(* CODESYS project sensores_v2_2_14.library
   Company: Teknike
   Version: 2.2.14
   DefaultNamespace: Teknike_Sensores
   Title: Sensores
   Placeholder: Teknike_Sensores
   Author: Tiago B. Cunico
   DocFormat: reStructuredText

Project tree, tasks and I/O mapping:
  libraries: BASIC, 3.31 (OSCAT); Tc2_ModbusRTU, * (Beckhoff Automation GmbH); Tc2_Standard, * (Beckhoff Automation GmbH); Tc2_System, * (Beckhoff Automation GmbH); Tc2_TcpIp, * (Beckhoff Automation GmbH); Tc2_Utilities, * (Beckhoff Automation GmbH); Tc3_Database, * (Beckhoff Automation GmbH); Tc3_Module, * (Beckhoff Automation GmbH); Geral, * (Teknike); TwinCAT Dynamic String Kit, * (FisoThemes)
  DUTs/
  Fbs/
    Analogica/
      Duts/
        data type Config_ST_SensorAnalogicos
        data type en_ST_SensorAnalogico
        data type sa_ST_SensorAnalogico
        data type st_SensorAnalogico
      function block FB_SensorAnalogico [ST]: AjeitaEntrada, AjeitaSaida
    Digital/
      SensorDigital/
        Duts/
          data type Config_ST_SensorDigital
          data type en_ST_SensorDigital
          data type ENUM_StatusSensor
          data type sa_ST_SensorDigital
          data type st_LeConfigSensorNoBanco
          data type st_SensorDigital
        function block FB_SensorDigital [ST]: FB_init, TamanhoCaixa
    Rede/
      322_485_Novus/
        Duts/
          data type entrada_N322_485_Novus
          data type Saida_N322_485_Novus
          data type st_N322_485_Novus
        function block N322_485_Novus [ST]
      RFID/
        function block FB_LeitorRFID_ViaOnda [ST]
        data type st_LeitorRFID_ViaOnda
      RTH_485_Novus/
        Duts/
          data type Config_RTH_485_Novus
          data type dt_RTH_485_Novus
          data type entrada_RTH_485_Novus
          data type Saida_RTH_485_Novus
        function block RTH_485_Novus [ST]
      SR2000/
        duts/
          data type ST_SR2000
          data type ST_SR2000_Config
          data type ST_SR2000_Entradas_Bloco
          data type ST_SR2000_Entradas_Dispositivo
          data type ST_SR2000_Saidas_Bloco
          data type ST_SR2000_Saidas_Dispositivo
        function F_AjeitaStringLeitor [ST]
        function block FB_SR2000 [ST]: AjustaEntrada, AjustaSaida, ContagemFalha, RequisitaDados, Status, TempoLeitura, TrabalhaResultado, Trigger
  GVLs/
    global variables GVL_Teste
  POUs/
    global variables GVL_BlibliotecaSensores
    program MAIN [ST]: ACT, Digital, SensorAnalogico
    program ValidaLicensa [ST]: Licensas
  Project Information/
    function F_GetCompany [ST]
    function F_GetTitle [ST]
    function F_GetVersion [ST]
  Version/
    global variables Global_Version
  VISUs/
*)

// Fbs/Analogica/Duts/Config_ST_SensorAnalogicos
TYPE Config_ST_SensorAnalogicos :
STRUCT PERSISTENT RETAIN
	rMinEntrada : REAL := 0; // valor minimo da entrada, normalmente 0
	rMaxEntrada : REAL := 32767; // valor maximo da entrada, normalmente 32767
	rMinSaida 	: REAL := 0; //minimo saida, normalmente 0
	rMaxSaida 	: REAL; // valor final, esse depende muito com o sensor
	iTempoFiltro: UDINT; // em ms
	sNome_Funcao: STRING;
	rOffset		: REAL; // offset direto na saida
		
	xForcaValor		: BOOL;				// ai ignora o valor que ta calculando e usa o valor que o cara setar
	rValorForcado	: REAL;				// valor que vai ser forçado
END_STRUCT
END_TYPE

// Fbs/Analogica/Duts/en_ST_SensorAnalogico
TYPE en_ST_SensorAnalogico :
	STRUCT
		iEntrada	: INT;	// valor vindo do sensor	
		i			: INT;	// Index para a IHM
	END_STRUCT
END_TYPE

// Fbs/Analogica/Duts/sa_ST_SensorAnalogico
TYPE sa_ST_SensorAnalogico :
	STRUCT
		rValor : REAL; // valor filtrado
		xPossivelFalha : BOOL; // se ficar mais de x tempo no no fim de escala ou no inicio dela é pq provavelmente deu pau
	END_STRUCT
END_TYPE

// Fbs/Analogica/Duts/st_SensorAnalogico
TYPE st_SensorAnalogico :
	STRUCT
		en		: en_ST_SensorAnalogico;
		config	: Config_ST_SensorAnalogicos;
		sa		: sa_ST_SensorAnalogico;
	END_STRUCT
END_TYPE

// Fbs/Digital/SensorDigital/Duts/Config_ST_SensorDigital
TYPE Config_ST_SensorDigital :
STRUCT RETAIN PERSISTENT
	xNF:		BOOL;
	rTmpOn:		REAL;
	rTmpOff:	REAL;
	sNome_Funcao: STRING;
END_STRUCT
END_TYPE

// Fbs/Digital/SensorDigital/Duts/en_ST_SensorDigital
TYPE en_ST_SensorDigital :
	STRUCT
		xSinalSensor	: BOOL;
		xResetContagem	: BOOL;
		i				: INT; // Index para a IHM	
		rVeloEsteira	: REAL;
	END_STRUCT
END_TYPE

// Fbs/Digital/SensorDigital/Duts/ENUM_StatusSensor
//{attribute 'qualified_only'}
//{attribute 'strict'}
TYPE ENUM_StatusSensor :
	(
		OBJETO_AUSENTE		:= 0,
		DETECTANDO_OBJETO	:= 1,
		OBJETO_PRESENTE		:= 2,
		DETECTANDO_AUSENCIA	:= 3
	);
END_TYPE

// Fbs/Digital/SensorDigital/Duts/sa_ST_SensorDigital
TYPE sa_ST_SensorDigital :
	STRUCT
		xObjPresente	: BOOL;
		uiContagem		: UINT;
		eStatus			: ENUM_StatusSensor;
		rTamanhoCaixa	: REAL; // tamanho da caixa em milimetros
	END_STRUCT
END_TYPE

// Fbs/Digital/SensorDigital/Duts/st_LeConfigSensorNoBanco
TYPE st_LeConfigSensorNoBanco :
	STRUCT
		Sensor		: T_ULARGE_INTEGER;
		Tag			: STRING(80);
		Funcao		: STRING(80);
		Timestamp	: DT;
	END_STRUCT
END_TYPE

// Fbs/Digital/SensorDigital/Duts/st_SensorDigital
TYPE st_SensorDigital :
	STRUCT
		en		: en_ST_SensorDigital;
		config	: Config_ST_SensorDigital;
		sa		: sa_ST_SensorDigital;
		Banco	: st_LeConfigSensorNoBanco;
	END_STRUCT
END_TYPE

// Fbs/Rede/322_485_Novus/Duts/entrada_N322_485_Novus
TYPE entrada_N322_485_Novus :
	STRUCT
		xComeca		: BOOL;
		iEndereco	: INT;	//endereço dele na rede
		i			: INT;	// Index para a IHM
		sNomeFuncao	: STRING;
		xForcaFalor : BOOL;
		rValorForcado : REAL;
		rOffset : REAL;
	END_STRUCT
END_TYPE

// Fbs/Rede/322_485_Novus/Duts/Saida_N322_485_Novus
TYPE Saida_N322_485_Novus :
	STRUCT
		xOcupado			: BOOL;
		xTerminei			: BOOL;
		rTemp				: REAL;
		xOnline				: BOOL;
		UltimoModbusErro	: MODBUS_ERRORS;
	END_STRUCT
END_TYPE

// Fbs/Rede/322_485_Novus/Duts/st_N322_485_Novus
TYPE st_N322_485_Novus :
	STRUCT
		en	: entrada_N322_485_Novus;
		sa	: Saida_N322_485_Novus;
	END_STRUCT
END_TYPE

// Fbs/Rede/RFID/st_LeitorRFID_ViaOnda
TYPE st_LeitorRFID_ViaOnda :
STRUCT
	xConecta : BOOL;	
	ip : T_IPv4Addr;
	xNovoResultado : BOOL;
	sTag : STRING;
	iTag : INT;
	xOnline : BOOL; //
END_STRUCT
END_TYPE

// Fbs/Rede/RTH_485_Novus/Duts/Config_RTH_485_Novus
TYPE Config_RTH_485_Novus :
STRUCT PERSISTENT RETAIN
	iEndereco 			: INT;
	iModoIndicacao		: INT;
	xUnidadeDeMedida	: BOOL;
	xBloqueiaConfigBT	: BOOL;
	rOffSetTemperatura	: REAL;
	rOffSetUmidade		: REAL;
	uiValorErro			: UINT;
END_STRUCT
END_TYPE

// Fbs/Rede/RTH_485_Novus/Duts/dt_RTH_485_Novus
TYPE dt_RTH_485_Novus :
	STRUCT
		en		: entrada_RTH_485_Novus;
		Config	: Config_RTH_485_Novus;
		sa		: Saida_RTH_485_Novus;
	END_STRUCT
END_TYPE

// Fbs/Rede/RTH_485_Novus/Duts/entrada_RTH_485_Novus
TYPE entrada_RTH_485_Novus :
	STRUCT
		xComeca			: BOOL;
		xEscreve		: BOOL;
		xAtualizaTudo	: BOOL;
		i				: INT; // Index para a IHM
	END_STRUCT
END_TYPE

// Fbs/Rede/RTH_485_Novus/Duts/Saida_RTH_485_Novus
TYPE Saida_RTH_485_Novus :
	STRUCT
		xTerminei : BOOL;

		rTemp					: REAL;
		rUmidade				: REAL;
		rPontoDeOrvalho			: REAL;
		iModoIndicacaoAtual		: INT;
		xUnidadeDeMedidaAtual	: BOOL;
		xHabilitaConfigBTAtual	: BOOL;
		rOffSetTemperaturaAtual	: REAL;
		rOffSetUmidadeAtual		: REAL;
		uiValorErroAtual		: UINT;
		xOnline					: BOOL;
		UltimoModbusErro		: ST_ModbusErrorDiagnostics;
	END_STRUCT
END_TYPE

// Fbs/Rede/SR2000/duts/ST_SR2000
TYPE ST_SR2000 :
	STRUCT
		En	: ST_SR2000_Entradas_Bloco;
		Sa	: ST_SR2000_Saidas_Bloco;
		Config : ST_SR2000_Config;
		

		En_D	AT %I*	: ST_SR2000_Entradas_Dispositivo;
		Sa_D	AT %Q*	: ST_SR2000_Saidas_Dispositivo;
	END_STRUCT
END_TYPE

// Fbs/Rede/SR2000/duts/ST_SR2000_Config
TYPE ST_SR2000_Config :
	STRUCT RETAIN PERSISTENT
		iIgnoraInicio : INT;
		iQuantosCharLe : INT;
	END_STRUCT
END_TYPE

// Fbs/Rede/SR2000/duts/ST_SR2000_Entradas_Bloco
TYPE ST_SR2000_Entradas_Bloco :
	STRUCT
		xLiga					: BOOL;
		xHabilitaAutoTrigger	: BOOL := true;
		xBtTriggerManual		: BOOL;
		xTrigManualCiclico		: BOOL;
		xSinalTrigAutomatico	: BOOL;
		xReset					: BOOL;
		sNome_Funcao			: STRING;
	END_STRUCT
END_TYPE

// Fbs/Rede/SR2000/duts/ST_SR2000_Entradas_Dispositivo
TYPE ST_SR2000_Entradas_Dispositivo :
	STRUCT

		State : UINT;

		xError					: BIT;
		xResultDataAvailable	: BIT;
		xResultDataStrobe		: BIT;

		xBufferOverflowError	: BIT;
		xGeneralError			: BIT;
		xBusy					: BIT;
		xTriggerBusy			: BIT;
		xLockBusy				: BIT;
		xModeBusy				: BIT;
		xErrBusy				: BIT;

		xREADY : BIT;

		xReadComplete				: BIT;
		xPresetComplete				: BIT;
		xRegisterPresetDataComplete	: BIT;
		xTuneComplete				: BIT;
		xBloadComplete				: BIT;

		xEXTRequestComplete			: BIT;
		xReadingFailure				: BIT;
		xPresetFailure				: BIT;
		xRegisterPresetDataFailure	: BIT;
		xTuneFailure				: BIT;
		xBloadFailure				: BIT;

		xEXTRequestFailure	: BIT;
		xIN1Status			: BIT;
		xIN2Status			: BIT;

		xOUT1Status	: BIT;
		xOUT2Status	: BIT;
		xOUT3Status	: BIT;

		xUnstable				: BIT;
		xMatchingLevelUnstable	: BIT;
		xISO_IEC15415Unstable	: BIT;
		xAIM_DPMUnstable		: BIT;
		xSAE_AS9132Unstable		: BIT;
		xISO_IEC15416Unstable	: BIT;

		uiMatchingLevel					: UINT;
		uiISO_IEC15415Grade				: UINT;
		uiAIM_DPMGrade					: UINT;
		uiISO_IEC15416Grade				: UINT;
		uiReadResultCode				: UINT;
		uiPresetResultCode				: UINT;
		uiRegisterPresetDataResultCode	: UINT;
		uiTuneResultCode				: UINT;
		uiBloadResultCode				: UINT;

		EXTRequestResultCode	: UINT;
		uiGeneralErrorCode		: UINT;
		uiSlaveID				: UINT;
		uiResultDataReadyCount	: UINT;
		uiResultDataUpdateCount	: UINT;
		uiMasterTriggerCount	: UINT;
		uiReadDataSize			: UINT;
		arResultData			: ARRAY[0..128] OF BYTE;

	END_STRUCT
END_TYPE

// Fbs/Rede/SR2000/duts/ST_SR2000_Saidas_Bloco
TYPE ST_SR2000_Saidas_Bloco :
	STRUCT

		xLeitorEmFalha	: BOOL;
		xLeitorPronto	: BOOL;
		xFalhaRede		: BOOL;
		ReadRequest		: BOOL;
		xNovoResultado	: BOOL;
		xFalhaLeitura	: BOOL;
		xNovosDados		: BOOL;
		sCodigoBruto	: STRING;
		sCodigo			: STRING;

		matchPorcentagem	: INT;
		NotaIsoIEC15415		: STRING;
		NotaIsoIEC15416		: STRING;
		NotaAimDPM			: STRING;

		uiTrigsTotais		: UINT;
		uiSucessoTotais		: UINT;
		uiFalhasTotais		: UINT;
		AcertoPorcentagem	: REAL;

		xSinalDeLiga : BOOL;
		
		sTempoTotalDeLeitura : STRING;
		sMediaTempoTotalDeLeitura : STRING;
	END_STRUCT
END_TYPE

// Fbs/Rede/SR2000/duts/ST_SR2000_Saidas_Dispositivo
TYPE ST_SR2000_Saidas_Dispositivo :
	STRUCT

		ctrl : UINT;

		ResultDataLatch				: BIT;
		ErrorClear					: BIT;
		ReadRequest					: BIT;
		PresetRequest				: BIT;
		RegisterPresetDataRequest	: BIT;
		TuneRequest					: BIT;
		BloadRequest				: BIT;

		ReadCompleteClear				: BIT;
		PresetCompleteClear				: BIT;
		RegisterPresetDataCompleteClear	: BIT;
		TuneCompleteClear				: BIT;
		BloadCompleteClear				: BIT;

		EXTRequestCompleteClear : BIT;

		BankNumber : UINT;

		UserDataSize	: UINT;
		UserData		: ARRAY[0..63] OF BYTE;
	END_STRUCT
END_TYPE

// GVLs/GVL_Teste
//{attribute 'qualified_only'}
VAR_GLOBAL PERSISTENT RETAIN

	stDigitaisss : st_SensorDigital;

	RTU : st_N322_485_Novus;

END_VAR

// POUs/GVL_BlibliotecaSensores
//{attribute 'qualified_only'}
VAR_GLOBAL
    {attribute 'hide'} 
	{attribute 'tc_no_symbol'}
	xLicensaValida1616848sdfs : BOOL;
	LicensaValida : BOOL;
	STCheckLicense : ST_CheckLicense;
END_VAR

// Version/Global_Version
{attribute 'TcGenerated'}
{attribute 'no-analysis'}
{attribute 'linkalways'}
// This function has been automatically generated from the project information.
VAR_GLOBAL CONSTANT
	{attribute 'const_non_replaced'}
	stLibVersion_Sensores : ST_LibVersion := (iMajor := 2, iMinor := 2, iBuild := 14, iRevision := 0, nFlags := 0, sVersion := '2.2.14');
END_VAR

// Fbs/Analogica/FB_SensorAnalogico
FUNCTION_BLOCK FB_SensorAnalogico
VAR_IN_OUT
	stAna : st_SensorAnalogico;
END_VAR
VAR_INPUT

	iEntrada		: INT;				// valor vindo do sensor	
	rMinEntrada		: REAL	:= 0;		// valor minimo da entrada, normalmente 0
	rMaxEntrada		: REAL	:= 32767;	// valor maximo da entrada, normalmente 32767
	rMinSaida		: REAL	:= 0;		// minimo saida, normalmente 0
	rMaxSaida		: REAL;				// valor final, esse depende muito com o sensor
	iTempoFiltro	: UDINT;			// em ms
	sNome_Funcao	: STRING;
	rOffset			: REAL; 			// offset direto na saida
	
	xForcaValor		: BOOL;				// ai ignora o valor que ta calculando e usa o valor que o cara setar
	rValorForcado	: REAL;				// valor que vai ser forçado

END_VAR
VAR_OUTPUT
	rValor : REAL; // valor filtrado
	xPossivelFalha : BOOL; // se ficar mais de x tempo no no fim de escala ou no inicio dela é pq provavelmente deu pau
END_VAR
VAR
	filtro	: BASIC.FT_PT1 (*Filter_PT1*) ;
	rAux	: REAL;
	
	tonFalha : TON;
	
	stAnaAnterior : st_SensorAnalogico;
END_VAR

IF xLicensaValida1616848sdfs THEN
	
	AjeitaEntrada();
	
	// transforma de inteiro pra real 
	rAux := BASIC.SCALE_R
		(
			X := iEntrada,
				I_LO := rMinEntrada,
				I_HI := rMaxEntrada,
				O_LO := rMinSaida,
				O_HI := rMaxSaida);
	
	// aplica um filtro de primeira ordem	
	
	//sanitizando entrada pra nao dar execção na bliblioteca do oscat
	IF iTempoFiltro < 5 AND iTempoFiltro <> 0 THEN
		filtro(in := rAux, T := UDINT_TO_TIME(0), K := 1, out => rValor);
	ELSE
		filtro(in := rAux, T := UDINT_TO_TIME(iTempoFiltro), K := 1, out => rValor);
	END_IF
	
	tonFalha(IN:= iEntrada = rMinEntrada OR iEntrada = rMaxEntrada, PT:= T#5M, Q=> xPossivelFalha, ET=> );
	
	rValor := rValor + rOffset;

	IF xForcaValor THEN
		rValor := rValorForcado;
	END_IF
	
	AjeitaSaida();
ELSE
	ValidaLicensa();
END_IF

ACTION AjeitaEntrada:





IF stAna.en.iEntrada <> stAnaAnterior.en.iEntrada THEN
	iEntrada := stAna.en.iEntrada;
END_IF
IF stAna.en.iEntrada <> iEntrada THEN
	stAna.en.iEntrada := iEntrada;
END_IF


IF stAna.config.rMinEntrada <> stAnaAnterior.config.rMinEntrada THEN
	rMinEntrada := stAna.config.rMinEntrada;
END_IF
IF stAna.config.rMinEntrada <> rMinEntrada THEN
	stAna.config.rMinEntrada := rMinEntrada;
END_IF


IF stAna.config.rMaxEntrada <> stAnaAnterior.config.rMaxEntrada THEN
	rMaxEntrada := stAna.config.rMaxEntrada;
END_IF
IF stAna.config.rMaxEntrada <> rMaxEntrada THEN
	stAna.config.rMaxEntrada := rMaxEntrada;
END_IF


IF stAna.config.rMinSaida <> stAnaAnterior.config.rMinSaida THEN
	rMinSaida := stAna.config.rMinSaida;
END_IF
IF stAna.config.rMinSaida <> rMinSaida THEN
	stAna.config.rMinSaida := rMinSaida;
END_IF


IF stAna.config.rMaxSaida <> stAnaAnterior.config.rMaxSaida THEN
	rMaxSaida := stAna.config.rMaxSaida;
END_IF
IF stAna.config.rMaxSaida <> rMaxSaida THEN
	stAna.config.rMaxSaida := rMaxSaida;
END_IF


IF stAna.config.iTempoFiltro <> stAnaAnterior.config.iTempoFiltro THEN
	iTempoFiltro := stAna.config.iTempoFiltro;
END_IF
IF stAna.config.iTempoFiltro <> iTempoFiltro THEN
	stAna.config.iTempoFiltro := iTempoFiltro;
END_IF


IF stAna.config.sNome_Funcao <> stAnaAnterior.config.sNome_Funcao THEN
	sNome_Funcao := stAna.config.sNome_Funcao;
END_IF
IF stAna.config.sNome_Funcao <> sNome_Funcao THEN
	stAna.config.sNome_Funcao := sNome_Funcao;
END_IF


IF stAna.config.rOffset <> stAnaAnterior.config.rOffset THEN
	rOffset := stAna.config.rOffset;
END_IF
IF stAna.config.rOffset <> rOffset THEN
	stAna.config.rOffset := rOffset;
END_IF


IF stAna.config.xForcaValor <> stAnaAnterior.config.xForcaValor THEN
	xForcaValor := stAna.config.xForcaValor;
END_IF
IF stAna.config.xForcaValor <> xForcaValor THEN
	stAna.config.xForcaValor := xForcaValor;
END_IF


IF stAna.config.rValorForcado <> stAnaAnterior.config.rValorForcado THEN
	rValorForcado := stAna.config.rValorForcado;
END_IF
IF stAna.config.rValorForcado <> rValorForcado THEN
	stAna.config.rValorForcado := rValorForcado;
END_IF



stAnaAnterior.en := stAna.en;
stAnaAnterior.config := stAna.config;
END_ACTION

ACTION AjeitaSaida:





stAna.sa.rValor := rValor;
stAna.sa.xPossivelFalha := xPossivelFalha;
END_ACTION

END_FUNCTION_BLOCK

// POUs/ValidaLicensa
PROGRAM ValidaLicensa
VAR
{attribute 'tc_no_symbol'}
Olhaliscensa : FB_CheckLicense;
{attribute 'tc_no_symbol'}
GUIDLicensa : GUID := STRING_TO_GUID('05F3F7DA-F1F3-425B-9124-1665F012FB6E');
END_VAR


Licensas();

STCheckLicense := Olhaliscensa.stCheckLicense;

xLicensaValida1616848sdfs :=
 Olhaliscensa.stCheckLicense.eResult = 0 OR //essa é so pros que sao da beckhoff mesmo
 Olhaliscensa.stCheckLicense.eResult = 16#203 OR
 Olhaliscensa.stCheckLicense.eResult = 16#254 OR
 Olhaliscensa.stCheckLicense.eResult = 16#255;

 LicensaValida := xLicensaValida1616848sdfs;

ACTION Licensas:
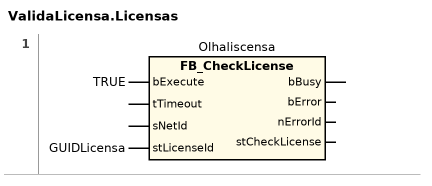
// NETWORK 1
Olhaliscensa(bExecute := TRUE, stLicenseId := GUIDLicensa); // FB_CheckLicense
END_ACTION

END_PROGRAM

// Fbs/Digital/SensorDigital/FB_SensorDigital
FUNCTION_BLOCK FB_SensorDigital
VAR_INPUT
	xSinalSensor	: BOOL;	(* sinal de campo do sensor *)
	xNF				: BOOL;	(* indica que o sensor tem lógica "presença de objeto em FALSE" *)
	rTmpOutOn		: REAL;	(* tempo de confirmação do sinal em ON *)
	rTmpOutOff		: REAL;	(* tempo de confirmação do sinal em OFF *)
	xResetContagem	: BOOL;	(* reset da contagem de pulsos de sensor *)
	sNome_Funcao	: STRING;
	rVeloEsteira	: REAL; // velocidade da esteira em que o sensor esta
END_VAR
VAR_OUTPUT
	xObjPresente	: BOOL;					(* indica presença de objeto *)
	uiContagem		: UINT;					(* contagem de objetos *)
	eStsSensor		: ENUM_StatusSensor;	(* status do sensor *)
	rTamanhoCaixa	: REAL; // tamanho em metros
END_VAR
VAR
	TON_TmrOutOn		: TON;
	TON_TmrOutOff		: TON;
	xSinalInternoSensor	: BOOL;
	RT_ObjetoPresente	: R_TRIG;
	
	//Pra ver o tamanho da caixa
	tInico 		: TIME;
	tFim		: TIME;
	tTotal 		: TIME;
	rtComeca	: R_TRIG;
	ftTermina	: f_TRIG;
END_VAR


IF xLicensaValida1616848sdfs THEN
		
	(* lógica de NA-NF *)
	IF xNF THEN
		xSinalInternoSensor := xSinalSensor = FALSE;
	ELSE
		xSinalInternoSensor := xSinalSensor = TRUE;
	END_IF
	
	(* definição de objeto presente *)
	IF TON_TmrOutOn.Q THEN
		xObjPresente := TRUE;
	END_IF
	
	IF TON_TmrOutOff.Q THEN
		xObjPresente := FALSE;
	END_IF
	
	TON_TmrOutOn(IN := xSinalInternoSensor, PT := REAL_TO_TIME(rTmpOutOn * 1000));
	TON_TmrOutOff(IN := NOT xSinalInternoSensor, PT := REAL_TO_TIME(rTmpOutOff * 1000));
	
	(* ao ligar a saída, incrementa a contagem de sensor *)
	RT_ObjetoPresente(CLK := xObjPresente);
	
	IF RT_ObjetoPresente.Q THEN
		uiContagem := uiContagem + 1;
	END_IF
	
	IF xResetContagem = TRUE THEN
		uiContagem := 0;
	END_IF
	
	(* status do sensor *)
	IF (NOT xSinalInternoSensor AND NOT xObjPresente) THEN
		eStsSensor := OBJETO_AUSENTE;
	END_IF (* ausência de objeto *)
	
	IF (xSinalInternoSensor AND NOT xObjPresente) THEN
		eStsSensor := DETECTANDO_OBJETO;
	END_IF (* presença de objeto em andamento *)
	
	IF (xSinalInternoSensor AND xObjPresente) THEN
		eStsSensor := OBJETO_PRESENTE;
	END_IF (* presença de objeto *)
	
	IF (NOT xSinalInternoSensor AND xObjPresente) THEN
		eStsSensor := DETECTANDO_AUSENCIA;
	END_IF (* ausência de objeto em andamento *)
	
	TamanhoCaixa();

ELSE
	ValidaLicensa();
END_IF

METHOD FB_init : BOOL
VAR_INPUT
	bInitRetains	: BOOL;	// if TRUE, the retain variables are initialized (warm start / cold start)
	bInCopyCode		: BOOL;	// if TRUE, the instance afterwards gets moved into the copy code (online change)
END_VAR

//Sanitizando entrada
IF xSinalSensor <> TRUE OR xSinalSensor <> FALSE THEN
	xSinalSensor := FALSE;
END_IF

IF xNF <> TRUE OR xNF <> FALSE THEN
	xNF := FALSE;
END_IF

IF rTmpOutOn < -0.1 OR rTmpOutOn > 3400000000000000000 THEN
	rTmpOutOn := 0;
END_IF

IF rTmpOutOff < -0.1 OR rTmpOutOff > 3400000000000000000 THEN
	rTmpOutOff := 0;
END_IF

IF xResetContagem <> TRUE OR xResetContagem <> FALSE THEN
	xResetContagem := FALSE;
END_IF
END_METHOD

ACTION TamanhoCaixa:



rtComeca(CLK:= xSinalSensor, Q=> );
IF rtComeca.q THEN
	tInico := TIME();
END_IF

ftTermina(CLK:= xSinalSensor, Q=> );
IF ftTermina.q THEN
	tFim := TIME();			// transforma pra milimetro por ms
	tTotal := tFim - tInico;//		1000 / 60 * 1000
	rTamanhoCaixa := rVeloEsteira * 0.0166666 * TIME_TO_UDINT(tTotal);
END_IF
END_ACTION

END_FUNCTION_BLOCK

// Fbs/Rede/322_485_Novus/N322_485_Novus
FUNCTION_BLOCK N322_485_Novus
VAR_IN_OUT
	MestreModbusRTU	: ModbusRtuMasterV2_KL6x22B;
	xComeca			: BOOL;
END_VAR
VAR_INPUT
	iEndereco : INT;
	xForcaFalor : BOOL;
	rValorForcado : REAL;
	rOffset : REAL;
END_VAR
VAR_OUTPUT
	xOcupado	: BOOL;
	xTerminei	: BOOL;
	rTemp		: REAL;
	xOnline		: BOOL;
	UltimoErro	: MODBUS_ERRORS;
END_VAR
VAR

	tonOnline	: ton;
	xAuxOnline	: BOOL;

	Registadores	: ARRAY[1..1] OF INT := [1];
	Valores			: ARRAY[1..1] OF UINT;

	timeoutvalue	: TIME := T#300MS;
	state			: INT;
	busy			: BOOL;

	iRegis			: INT	:= 1;
	iRegisEscrita	: INT	:= 1;

	rAux : REAL;

	rtComeca : R_TRIG;

	i : INT;

	xEscreveInterno		: BOOL;
	rtEscreveInterno	: R_TRIG;

	xAtualizaTudoInterno	: BOOL;
	rtAtualizaTudoInterno	: R_TRIG;

END_VAR

// caso voce esteja com problema em que ele funciona de vez em quando ou da erro no CRC ou mesmo invalid operation
// vale lembrar que precisa ativar ele pra half duplex e ficar em 8N1
// eu ja perdi algumas horas com esse problema, vc nao precisa tb
// vai la meu guerrerinho

IF xLicensaValida1616848sdfs THEN
	
	xTerminei := FALSE;
	
	rtComeca(CLK := xComeca, Q =>);
	
	IF rtComeca.q THEN
		xAuxOnline := FALSE;
	END_IF
	
	CASE state OF
	
		0:
			// ele so mexe no mestre caso seja a vez dele
			IF xComeca THEN
				MestreModbusRTU.ReadRegs(Execute := FALSE); //bota em 0 pra reiniciar	
				state := 1;
			END_IF
	
		1: //Le registradores
			MestreModbusRTU.ReadRegs
				(
					UnitID := TO_BYTE(iEndereco),
						Quantity := 1,
						MBAddr := TO_WORD(Registadores[1]),
						cbLength := SIZEOF(Valores[1]),
						pMemoryAddr := ADR(Valores[1]),
						Execute := TRUE,
						Timeout := timeoutvalue,
						Busy => busy);
	
			IF NOT busy THEN
				MestreModbusRTU.ReadRegs(Execute := FALSE);
				// so fica online se ler tudo e nenhumm der erro
				xAuxOnline := MestreModbusRTU.Error;
				// joga de volta pro 0 pra ver se ele terminou
				state		:= 0;
				xTerminei	:= TRUE;
				xComeca		:= FALSE;
			END_IF
	
	END_CASE
	
	tonOnline(IN := NOT xAuxOnline, PT := T#0.5S, Q =>, ET =>);
	xOnline := tonOnline.q;
	
	UltimoErro := MestreModbusRTU.ErrorDiagnostics.LastErrorID;
	
	xOcupado := MestreModbusRTU.BUSY AND xComeca;
	
	rAux	:= TO_INT(Valores[1]);
	rTemp	:= rAux / 10;
	rTemp	:= rTemp + rOffset;
	
	IF xForcaFalor THEN
		rTemp := rValorForcado;
	END_IF
	
ELSE
	ValidaLicensa();
END_IF

END_FUNCTION_BLOCK

// Fbs/Rede/RFID/FB_LeitorRFID_ViaOnda
//{attribute 'hide_all_locals'}
FUNCTION_BLOCK FB_LeitorRFID_ViaOnda
VAR_INPUT
	xConecta : BOOL := TRUE;	
	ip : T_IPv4Addr := '192.168.100.20';
END_VAR
VAR_OUTPUT
	xNovoResultado : BOOL;
	sTag : STRING;
	iTag : INT;
	xOnline : BOOL; //
END_VAR
VAR	
	xAmostra : BOOL;

	fbConection : FB_ClientServerConnection;
	fbRecebe : FB_SocketReceive;
	sRecebido: STRING(1000);
	sRecebidoB: STRING(1000);
	rtTerminouDeMandarOComando : R_TRIG;
	tPeraUmPoucoAntesDePedirOqueVeio : TON;
	xManda: BOOL;
	tEspera : TIME;
	rtAmostra : R_TRIG;
	
	fbSB : FB_StringBuilder;
	fbSBaux : FB_StringBuilder;
	


END_VAR



xNovoResultado := FALSE;



//conecta na tcp socket
fbConection(
	sSrvNetID:= '', 
	nMode:= CONNECT_MODE_ENABLEDBG, 
	sRemoteHost:= ip, 
	nRemotePort:= 5000, 
	bEnable:= xConecta, 
	tReconnect:= T#5S, 
	bBusy=> , 
	bError=> , 
	nErrId=> , 
	hSocket=> , 
	eState=> );
	


//fica rodando o recebe pra ficar lendo caso aparece alguma coisa
IF NOT fbRecebe.bExecute THEN
	fbRecebe.bExecute := TRUE;
END_IF
	
fbRecebe(
	sSrvNetId:= '', 
	hSocket:= fbConection.hSocket, 
	cbLen:= SIZEOF(sRecebidoB), 
	pDest:= ADR(sRecebidoB), 
	bExecute:= , 
	tTimeout:= , 
	bBusy=> , 
	bError=> , 
	nErrId=> , 
	nRecBytes=> );
	
IF NOT fbRecebe.bBusy THEN
		
	IF fbRecebe.nRecBytes > 0 THEN
		//ajusta o que veio pra ficar como a gente quer
		sRecebido := LEFT(STR:= sRecebidoB, SIZE:=TO_INT(fbRecebe.nRecBytes));
		
		fbSB.Clear();
		fbSB.Append(sRecebido);
		fbSB.Replace('$$','',TRUE);
		fbSB.Replace('$$R$$N','',TRUE);
						 
		sRecebido := fbSB.GetString();
		
		IF sRecebido <> 'FAIL' OR  sRecebido <> 'STOPOK' OR  sRecebido <> 'STARTOK' THEN
			sTag := sRecebido;
			iTag := STRING_TO_INT(sTag);
		END_IF
		
		xNovoResultado := TRUE;
	
	END_IF
	
	fbRecebe.bExecute := FALSE;
	fbRecebe();
	
END_IF

END_FUNCTION_BLOCK

// Fbs/Rede/RTH_485_Novus/RTH_485_Novus
FUNCTION_BLOCK RTH_485_Novus
VAR_IN_OUT
	MestreModbusRTU : ModbusRtuMasterV2_KL6x22B;
END_VAR
VAR_INPUT

	xComeca			: BOOL;
	xEscreve		: BOOL;
	xAtualizaTudo	: BOOL;

	iEndereco			: INT;
	iModoIndicacao		: INT;
	xUnidadeDeMedida	: BOOL;
	xBloqueiaConfigBT	: BOOL;
	rOffSetTemperatura	: REAL;
	rOffSetUmidade		: REAL;
	uiValorErro			: UINT;
END_VAR
VAR_OUTPUT
	xTerminei : BOOL;

	rTemp					: REAL;
	rUmidade				: REAL;
	rPontoDeOrvalho			: REAL;
	iModoIndicacaoAtual		: INT;
	xUnidadeDeMedidaAtual	: BOOL;
	xHabilitaConfigBTAtual	: BOOL;
	rOffSetTemperaturaAtual	: REAL;
	rOffSetUmidadeAtual		: REAL;
	uiValorErroAtual		: UINT;
	xOnline					: BOOL;
	UltimoModbusErro		: ST_ModbusErrorDiagnostics;
END_VAR
VAR

	tonOnline	: ton;
	xAuxOnline	: BOOL;

	Registadores : ARRAY[1..10] OF INT := [5,6,7,8,9,10,11,12,14,16];

	Valores : ARRAY[1..10] OF UINT;

	RegistadoresEscrita : ARRAY[1..6] OF INT := [6,10,11,12,14,16];

	ValoresEscrita		: ARRAY[1..10] OF UINT;
	xTerminouEscrever	: BOOL;

	timeoutvalue	: TIME := T#300MS;
	state			: INT;
	busy			: BOOL;

	iRegis			: INT	:= 1;
	iRegisEscrita	: INT	:= 1;

	rAux : REAL;

	rtComeca : R_TRIG;

	i : INT;

	xEscreveInterno		: BOOL;
	rtEscreveInterno	: R_TRIG;

	xAtualizaTudoInterno	: BOOL;
	rtAtualizaTudoInterno	: R_TRIG;

END_VAR


IF xLicensaValida1616848sdfs THEN	
	
	rtComeca(CLK := xComeca, Q =>);
	
	IF rtComeca.q THEN
		xTerminei := FALSE;
	
		IF xAtualizaTudoInterno THEN
			iRegis := 1;
		ELSE
			iRegis := 3;
		END_IF
	
		iRegisEscrita	:= 1;
		xAuxOnline		:= FALSE;
	END_IF
	
	rtEscreveInterno(CLK := xEscreve, Q =>);
	
	IF rtEscreveInterno.q THEN
		xEscreveInterno := TRUE;
	END_IF
	
	rtAtualizaTudoInterno(CLK := xAtualizaTudo, Q =>);
	
	IF rtAtualizaTudoInterno.q THEN
		xAtualizaTudoInterno := TRUE;
	END_IF
	
	//Joga valores de escrita no vetor
	ValoresEscrita[1]	:= TO_UINT(iModoIndicacao);
	ValoresEscrita[2]	:= TO_UINT(xUnidadeDeMedida);
	ValoresEscrita[3]	:= TO_UINT(xBloqueiaConfigBT);
	ValoresEscrita[4]	:= TO_UINT(rOffSetTemperatura * 10);
	ValoresEscrita[5]	:= TO_UINT(rOffSetUmidade * 10);
	ValoresEscrita[6]	:= uiValorErro;
	
	CASE state OF
	
		0:
			// ele so mexe no mestre caso seja a vez dele
			IF xComeca AND NOT xTerminei THEN
				MestreModbusRTU.ReadRegs(Execute := FALSE); //bota em 0 pra reiniciar
			END_IF
	
			// ele vai tentar ir ate 10 caso esteja liberado, se nao vai so ate 5
			IF (xAtualizaTudoInterno AND iRegis < 11) OR (NOT xAtualizaTudoInterno AND iRegis < 6) THEN
				state := 1;
			ELSE
				// se tiver que escrever ele vai pra parte de escrita se nao ele terminou
				IF (xEscreveInterno AND iRegisEscrita > 6) OR NOT xEscreveInterno THEN
					xTerminei				:= TRUE;
					xEscreveInterno			:= FALSE;
					xAtualizaTudoInterno	:= false;
					state					:= 0;
				ELSE
					state := 2;
				END_IF
	
			END_IF
	
		1: //Le registradores
			MestreModbusRTU.ReadRegs
				(
					UnitID := TO_BYTE(iEndereco),
						Quantity := 1,
						MBAddr := TO_WORD(Registadores[iRegis]),
						cbLength := SIZEOF(Valores[iRegis]),
						pMemoryAddr := ADR(Valores[iRegis]),
						Execute := TRUE,
						Timeout := timeoutvalue,
						Busy => busy);
	
			IF NOT busy THEN
				MestreModbusRTU.ReadRegs(Execute := FALSE);
				// so fica online se ler tudo e nenhumm der erro
				xAuxOnline := xAuxOnline OR MestreModbusRTU.Error;
				// joga de volta pro 0 pra ver se ele terminou
				state := 0;
				// vai para o proximo registrador
				iRegis := iRegis + 1;
			END_IF
	
		2: //escreve no registrador
			MestreModbusRTU.WriteSingleRegister
				(
					UnitID := TO_BYTE(iEndereco),
						Quantity := 1,
						MBAddr := TO_WORD(RegistadoresEscrita[iRegisEscrita]),
						cbLength := SIZEOF(ValoresEscrita[iRegisEscrita]),
						pMemoryAddr := ADR(ValoresEscrita[iRegisEscrita]),
						Execute := TRUE,
						Timeout := timeoutvalue,
						Busy => busy);
	
			IF NOT busy THEN
				MestreModbusRTU.WriteSingleRegister(Execute := FALSE);
				state			:= 0;
				iRegisEscrita	:= iRegisEscrita + 1;
			END_IF
	END_CASE
	
	// um filtrinho caso ele nao consiga ler um registrador e de erro
	IF xTerminei THEN
		tonOnline(IN := xAuxOnline, PT := T#1S, Q =>, ET =>);
		xOnline := NOT tonOnline.Q;
	END_IF
	
	tonOnline();
	
	UltimoModbusErro := MestreModbusRTU.ErrorDiagnostics;
	
	iModoIndicacaoAtual := TO_INT(Valores[2]);
	
	rAux	:= TO_INT(Valores[3]);
	rTemp	:= rAux / 10;
	
	rAux		:= TO_INT(Valores[4]);
	rUmidade	:= rAux / 10;
	
	rAux			:= TO_INT(Valores[5]);
	rPontoDeOrvalho	:= rAux / 10;
	
	xUnidadeDeMedidaAtual	:= TO_BOOL(Valores[6]);
	xHabilitaConfigBTAtual	:= TO_BOOL(Valores[7]);
	
	rAux					:= TO_INT(Valores[8]);
	rOffSetTemperaturaAtual	:= (rAux) / 10;
	
	rAux				:= TO_INT(Valores[9]);
	rOffSetUmidadeAtual	:= (rAux) / 10;
	
	uiValorErroAtual := (Valores[10]);

ELSE
	ValidaLicensa();
END_IF

END_FUNCTION_BLOCK

// Fbs/Rede/SR2000/F_AjeitaStringLeitor
FUNCTION F_AjeitaStringLeitor : String
VAR_INPUT
	Entrada : STRING;
	iIgnoraInicio : INT;
	iQuantosCharLe : INT;
END_VAR
VAR
END_VAR



F_AjeitaStringLeitor := DELETE(STR:=Entrada , LEN:= iIgnoraInicio+1,POS:=0 );

F_AjeitaStringLeitor := LEFT(STR:= F_AjeitaStringLeitor, SIZE:= iQuantosCharLe);

END_FUNCTION

// Fbs/Rede/SR2000/FB_SR2000
FUNCTION_BLOCK FB_SR2000
VAR_IN_OUT
	st_SR2000 : ST_SR2000;
END_VAR
VAR_INPUT
	xLiga					: BOOL;
	xHabilitaAutoTrigger	: BOOL;
	xBtTriggerManual		: BOOL;
	xTrigManualCiclico		: BOOL;
	xSinalTrigAutomatico	: BOOL;
	xReset					: BOOL;
	
	iIgnoraInicio : INT;
	iQuantosCharLe : INT;
	rTempoTrig : REAL;
END_VAR
VAR_OUTPUT
	xLeitorEmFalha	: BOOL;
	xLeitorPronto	: BOOL;
	xFalhaRede		: BOOL;
	ReadRequest		: BOOL;
	xNovoResultado	: BOOL;
	xNovosDados		: BOOL;
	xFalhaLeitura	: BOOL;
	sCodigoBruto	: STRING;
	sCodigo			: STRING;

	matchPorcentagem	: INT;
	NotaIsoIEC15415		: STRING;	// valido para QR code
	NotaIsoIEC15416		: STRING;	// valido para codigo de barras
	NotaAimDPM			: STRING;	// valido para QR code

	uiTrigsTotais		: UINT;
	uiSucessoTotais		: UINT;
	uiFalhasTotais		: UINT;
	AcertoPorcentagem	: REAL;

	xSinalDeLiga : BOOL;
	
	sTempoTotalDeLeitura : STRING;	
	sMediaTempoTotalDeLeitura : STRING;
END_VAR
VAR
	ultimo_st_SR2000	: ST_SR2000;
	xNovaRequest		: BOOL;
	rtNovaRequest		: R_TRIG;
	rtNovaRequest2		: R_TRIG;
	rtNovaResultado		: R_TRIG;
	rtNovosDados		: R_TRIG;
	tonTrigCiclico		: TON;
	rtRequest			: R_TRIG;
	xAuxRquest			: BOOL;

	xRequesitaDados					: BOOL;
	uiResultDataUpdateCountAnterior	: UINT;

	contadorErro	: CTU;
	rAux			: REAL;
	
	rtComecouLeitura : R_TRIG;
	rtTerminouLeitura : R_TRIG;
	TonLeitura : TON;
	
	tMedia : ARRAY[1..20] OF TIME;
	i : INT;
	tSoma : TIME;
	tonTimeOut : TON;
END_VAR


IF xLicensaValida1616848sdfs THEN	

	xSinalDeLiga := xLiga;
	
	AjustaEntrada();
	
	Status();
	
	Trigger();
	
	RequisitaDados();
	
	TrabalhaResultado();
	
	ContagemFalha();
	
	TempoLeitura();
	
	AjustaSaida();
	
ELSE
	ValidaLicensa();
END_IF

ACTION AjustaEntrada:


IF st_SR2000.Config.iIgnoraInicio <> ultimo_st_SR2000.Config.iIgnoraInicio THEN
	iIgnoraInicio := st_SR2000.Config.iIgnoraInicio;
END_IF

IF st_SR2000.Config.iQuantosCharLe <> ultimo_st_SR2000.Config.iQuantosCharLe THEN
	iQuantosCharLe := st_SR2000.Config.iQuantosCharLe;
END_IF


IF st_SR2000.En.xHabilitaAutoTrigger <> ultimo_st_SR2000.En.xHabilitaAutoTrigger THEN
	xHabilitaAutoTrigger := st_SR2000.En.xHabilitaAutoTrigger;
END_IF

IF xHabilitaAutoTrigger <> ultimo_st_SR2000.En.xHabilitaAutoTrigger THEN
	st_SR2000.En.xHabilitaAutoTrigger := xHabilitaAutoTrigger;
END_IF

IF st_SR2000.En.xBtTriggerManual <> ultimo_st_SR2000.En.xBtTriggerManual THEN
	xBtTriggerManual := st_SR2000.En.xBtTriggerManual;
END_IF

IF xBtTriggerManual <> ultimo_st_SR2000.En.xBtTriggerManual THEN
	st_SR2000.En.xBtTriggerManual := xBtTriggerManual;
END_IF

IF st_SR2000.En.xSinalTrigAutomatico <> ultimo_st_SR2000.En.xSinalTrigAutomatico THEN
	xSinalTrigAutomatico := st_SR2000.En.xSinalTrigAutomatico;
END_IF

IF xSinalTrigAutomatico <> ultimo_st_SR2000.En.xSinalTrigAutomatico THEN
	st_SR2000.En.xSinalTrigAutomatico := xSinalTrigAutomatico;
END_IF

IF st_SR2000.En.xReset <> ultimo_st_SR2000.En.xReset THEN
	xReset := st_SR2000.En.xReset;
END_IF

IF xReset <> ultimo_st_SR2000.En.xReset THEN
	st_SR2000.En.xReset := xReset;
END_IF

IF st_SR2000.En.xTrigManualCiclico <> ultimo_st_SR2000.En.xTrigManualCiclico THEN
	xTrigManualCiclico := st_SR2000.En.xTrigManualCiclico;
END_IF

IF xTrigManualCiclico <> ultimo_st_SR2000.En.xTrigManualCiclico THEN
	st_SR2000.En.xTrigManualCiclico := xTrigManualCiclico;
END_IF

IF st_SR2000.En.xLiga <> ultimo_st_SR2000.En.xLiga THEN
	xSinalDeLiga := st_SR2000.En.xLiga;
END_IF

IF xLiga <> ultimo_st_SR2000.En.xLiga THEN
	st_SR2000.En.xLiga := xLiga;
END_IF

IF iIgnoraInicio <> ultimo_st_SR2000.Config.iIgnoraInicio THEN
	st_SR2000.Config.iIgnoraInicio := iIgnoraInicio;
END_IF

IF iQuantosCharLe <> ultimo_st_SR2000.Config.iQuantosCharLe THEN
	st_SR2000.Config.iQuantosCharLe := iQuantosCharLe;
END_IF

ultimo_st_SR2000 := st_SR2000;
END_ACTION

ACTION AjustaSaida:

st_SR2000.Sa.xLeitorPronto			:= xLeitorPronto;
st_SR2000.Sa.xFalhaRede				:= xFalhaRede;
st_SR2000.Sa.ReadRequest			:= ReadRequest;	//sinal pra fora
st_SR2000.Sa_D.ReadRequest			:= ReadRequest;	//sinal pro leitor
st_SR2000.Sa_D.ReadCompleteClear	:= ReadRequest;	//limpa o status de nova leitura
st_SR2000.Sa.xNovoResultado			:= xNovoResultado;
st_SR2000.Sa.xNovosDados			:= xNovosDados;
st_SR2000.Sa.sCodigoBruto			:= sCodigoBruto;
st_SR2000.Sa.sCodigo 				:= sCodigo;
st_SR2000.Sa_D.ErrorClear			:= xReset; //limpa o s

st_SR2000.Sa_D.ResultDataLatch := xRequesitaDados;

st_SR2000.Sa.matchPorcentagem	:= matchPorcentagem;
st_SR2000.Sa.NotaIsoIEC15415	:= NotaIsoIEC15415;
st_SR2000.Sa.NotaIsoIEC15416	:= NotaIsoIEC15416;
st_SR2000.Sa.NotaAimDPM			:= NotaAimDPM;

st_SR2000.Sa.xLeitorEmFalha := xLeitorEmFalha;

st_SR2000.Sa.uiFalhasTotais		:= uiFalhasTotais;
st_SR2000.Sa.uiSucessoTotais	:= uiSucessoTotais;
st_SR2000.Sa.uiTrigsTotais		:= uiTrigsTotais;
st_SR2000.Sa.AcertoPorcentagem	:= AcertoPorcentagem;

st_SR2000.Sa.sTempoTotalDeLeitura := sTempoTotalDeLeitura;
END_ACTION

ACTION ContagemFalha:

contadorErro
	(
		CU := st_SR2000.En_D.xReadingFailure,
			RESET := contadorErro.CV > st_SR2000.En_D.uiResultDataReadyCount,
			PV :=,
			Q =>,
			CV =>);
END_ACTION

ACTION RequisitaDados:

IF st_SR2000.En_D.uiResultDataReadyCount <> st_SR2000.En_D.uiResultDataUpdateCount AND st_SR2000.En_D.xResultDataAvailable THEN
	IF uiResultDataUpdateCountAnterior = st_SR2000.En_D.uiResultDataUpdateCount THEN
		xRequesitaDados := TRUE;
	ELSE
		uiResultDataUpdateCountAnterior	:= st_SR2000.En_D.uiResultDataUpdateCount;
		xRequesitaDados					:= FALSE;
	END_IF
ELSE
	xRequesitaDados	:= FALSE;
	xNovosDados		:= FALSE;

	IF NOT st_SR2000.En_D.xResultDataAvailable THEN
		uiResultDataUpdateCountAnterior := st_SR2000.En_D.uiResultDataUpdateCount;
	ELSE
		xNovosDados := TRUE;
	END_IF
END_IF
END_ACTION

ACTION Status:

xLeitorPronto	:= st_SR2000.En_D.xREADY;
xFalhaRede		:= st_SR2000.En_D.State <> 0;

xNovoResultado	:= (st_SR2000.En_D.xReadComplete AND NOT st_SR2000.En_D.xResultDataAvailable) OR st_SR2000.En_D.xReadingFailure;
xFalhaLeitura	:= st_SR2000.En_D.xReadingFailure;

xLeitorEmFalha := st_SR2000.En_D.xError;

uiTrigsTotais	:= st_SR2000.En_D.uiMasterTriggerCount;
uiSucessoTotais	:= st_SR2000.En_D.uiMasterTriggerCount - contadorErro.CV;
uiFalhasTotais	:= contadorErro.cv;

rAux := uiSucessoTotais;

IF uiTrigsTotais <> 0 THEN
	rAux := rAux * 100 / uiTrigsTotais;
END_IF

AcertoPorcentagem := rAux;

IF xNovoResultado THEN
	matchPorcentagem := UINT_TO_INT(st_SR2000.En_D.uiMatchingLevel);

	CASE st_SR2000.En_D.uiISO_IEC15415Grade OF

		0:
			NotaIsoIEC15415 := 'E';

		1:
			NotaIsoIEC15415 := 'D';

		2:
			NotaIsoIEC15415 := 'C';

		3:
			NotaIsoIEC15415 := 'B';

		4:
			NotaIsoIEC15415 := 'A';
	END_CASE

	CASE st_SR2000.En_D.uiISO_IEC15416Grade OF

		0:
			NotaIsoIEC15416 := 'E';

		1:
			NotaIsoIEC15416 := 'D';

		2:
			NotaIsoIEC15416 := 'C';

		3:
			NotaIsoIEC15416 := 'B';

		4:
			NotaIsoIEC15416 := 'A';
	END_CASE

	CASE st_SR2000.En_D.uiAIM_DPMGrade OF

		0:
			NotaAimDPM := 'E';

		1:
			NotaAimDPM := 'D';

		2:
			NotaAimDPM := 'C';

		3:
			NotaAimDPM := 'B';

		4:
			NotaAimDPM := 'A';
	END_CASE
END_IF
END_ACTION

ACTION TempoLeitura:


rtComecouLeitura(CLK:= ReadRequest, Q=> );
IF rtComecouLeitura.q THEN
	TonLeitura.IN := TRUE;
END_IF

TonLeitura(PT:=T#1H , Q=> , ET=> );

rtTerminouLeitura(CLK:= xNovoResultado OR st_SR2000.En_D.xReadingFailure, Q=> );
IF rtTerminouLeitura.q THEN
	TonLeitura.IN := FALSE;
	sTempoTotalDeLeitura := F_TempoEmStringAteHoras(Tempo:= TonLeitura.ET, 
													xMostraHoras:= FALSE, 
													xMostraMinutos:= FALSE, 
													xMostraSegundos:= TRUE, 
													xMostraMilisegundos:= TRUE, 
													xCascata:= TRUE);
													
	FOR i := 20 TO 2 BY -1 DO
		tMedia[i] := tMedia[i + 1];
	END_FOR
	
	tMedia[1] := TonLeitura.ET;
	
	tSoma := T#0S;
	FOR i := 1 TO 20 DO
		IF tMedia[i] > T#0S THEN	
			tSoma := tSoma + tMedia[i];
		END_IF
	END_FOR
	
	IF I < 2  THEN
		i := 2;
	END_IF
	
	sMediaTempoTotalDeLeitura := F_TempoEmStringAteHoras(Tempo:= tSoma/(i-1), 
															xMostraHoras:= FALSE, 
															xMostraMinutos:= FALSE, 
															xMostraSegundos:= TRUE, 
															xMostraMilisegundos:= TRUE, 
															xCascata:= TRUE);									
END_IF
END_ACTION

ACTION TrabalhaResultado:

IF xNovosDados THEN

	IF NOT xFalhaLeitura THEN
		sCodigoBruto := '';

		MEMMOVE
			(
				srcAddr := ADR(st_SR2000.En_D.arResultData),
					destAddr := ADR(sCodigoBruto),
					n := st_SR2000.En_D.uiReadDataSize);
					
		sCodigo := F_AjeitaStringLeitor(Entrada:= sCodigoBruto, iIgnoraInicio:= iIgnoraInicio, iQuantosCharLe:= iQuantosCharLe);
	ELSE
		sCodigoBruto := sCodigo := '--NoREAD';
	END_IF
END_IF
END_ACTION

ACTION Trigger:


// se for em manual ele tira de true o sinal pra ficar mais facil
rtNovaRequest(CLK := st_SR2000.En_D.xReadComplete OR st_SR2000.En_D.xReadingFailure, Q =>);
//rtNovaRequest2(CLK := NOT st_SR2000.En_D.xTriggerBusy, Q =>);

IF rtNovaRequest.q  OR rtNovaRequest2.q THEN
	ReadRequest			:= FALSE;
	xBtTriggerManual	:= FALSE;
	xAuxRquest			:= false;
END_IF
// faz uma nova leitura e limpa o estatus de leitura feita


IF xHabilitaAutoTrigger THEN
	xAuxRquest := xSinalTrigAutomatico;
ELSE
	IF xTrigManualCiclico THEN
		tonTrigCiclico.IN := TRUE;

		IF tonTrigCiclico.q THEN
			xAuxRquest			:= TRUE;
			tonTrigCiclico.IN	:= FALSE;
		END_IF

		tonTrigCiclico(IN :=, PT := T#1S, Q =>, ET =>);
	ELSE
		xAuxRquest := xBtTriggerManual;
	END_IF
END_IF

rtRequest(CLK := xAuxRquest, Q =>);

IF rtRequest.q THEN
	ReadRequest := TRUE;
END_IF


tonTimeOut(IN:= ReadRequest, PT:=REAL_TO_TIME(rTempoTrig*1000), Q=> , ET=> );
IF tonTimeOut.q THEN
	ReadRequest := FALSE;
END_IF
END_ACTION

END_FUNCTION_BLOCK

// POUs/MAIN
PROGRAM MAIN
VAR

	stSR2000 : ST_SR2000;
	fbSR2000 : FB_SR2000;
	fbDigital : FB_SensorDigital;
	fbAnalogico : FB_SensorAnalogico;
	
	tonAux : TON;
	

	xfirstScan : BOOL := TRUE;
	
	stAnalogica : st_SensorAnalogico;
	FBViaOnda : FB_LeitorRFID_ViaOnda;

END_VAR

//ACT();

IF tonAux.Q THEN
	tonAux(IN := false);
END_IF
tonAux(IN := TRUE);

fbDigital.xSinalSensor := NOT tonAux.Q;

Digital();

SensorAnalogico();

ACTION ACT:
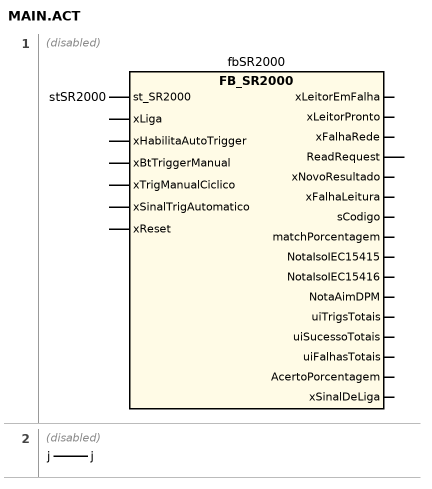
// NETWORK 1 (disabled)
// fbSR2000(st_SR2000 := stSR2000); // FB_SR2000

// NETWORK 2 (disabled)
// j := j;
END_ACTION

ACTION Digital:
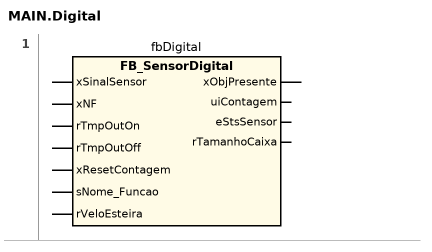
// NETWORK 1
fbDigital(); // FB_SensorDigital
END_ACTION

ACTION SensorAnalogico:
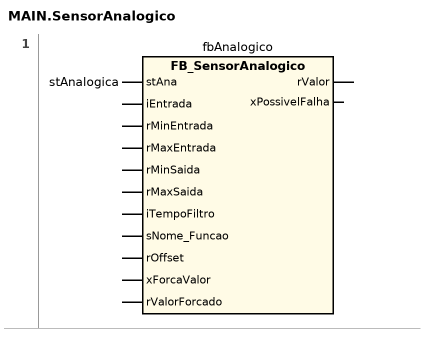
// NETWORK 1
fbAnalogico(stAna := stAnalogica); // FB_SensorAnalogico
END_ACTION

END_PROGRAM

// Project Information/F_GetCompany
// This function has been automatically generated from the project information.
{attribute 'signature_flag' := '1073741824'}
{attribute 'TcGenerated'}
{attribute 'no-analysis'}
FUNCTION F_GetCompany : WSTRING
VAR_INPUT
	
END_VAR

F_GetCompany := "Teknike";

END_FUNCTION

// Project Information/F_GetTitle
// This function has been automatically generated from the project information.
{attribute 'signature_flag' := '1073741824'}
{attribute 'TcGenerated'}
{attribute 'no-analysis'}
FUNCTION F_GetTitle : WSTRING
VAR_INPUT
	
END_VAR

F_GetTitle := "Sensores";

END_FUNCTION

// Project Information/F_GetVersion
// This function has been automatically generated from the project information.
{attribute 'signature_flag' := '1073741824'}
{attribute 'TcGenerated'}
{attribute 'no-analysis'}
FUNCTION F_GetVersion : ST_LibVersion
VAR_INPUT
	
END_VAR

F_GetVersion.iMajor := 2;
F_GetVersion.iMinor := 2;
F_GetVersion.iBuild := 14;
F_GetVersion.iRevision := 0;
F_GetVersion.sVersion := '2.2.14';
F_GetVersion.nFlags := 0;

END_FUNCTION
